SUBAPPLICATION NumericValue_TO_AR2_OPC (* VT-Eingabefeld (CInputNumber) UND OPC-UA (Remote) lesen, letzter Schreiber gewinnt (AR_LAST_2), als AR2 (bidirektional) an einen Consumer weiterreichen. Was der Consumer zurueckechot wird auf BEIDE Wege zurueckgemeldet (VT-Anzeige + Publish) *)
  (* Standard: 61499-2; Description: Copyright (c) 2026 Meisterschulen am Ostbahnhof This program and the accompanying materials are made available under the terms of the Eclipse Public License 2.0 which is available at https://www.eclipse.org/legal/epl-2.0/ SPDX-License-Identifier: EPL-2.0 *)
  (* Version 1.1, 2026-09-16, Franz Höpfinger, Meisterschulen am Ostbahnhof, Neuer optionaler Ausgangs-Plug VALUE_OUT ergaenzt (AR_SPLIT_2 zu AR_SPLIT_3, 3. Zweig = plain-AR-Spiegel von AR_TO_AR2.AR_OUT) - damit externe Consumer den aktuellen Wert lesen koennen, ohne selbst denselben OPC-UA-Knoten lokal zu abonnieren (FORTE: 'Cannot add another one'). Unverdrahtet lassen, wenn nicht gebraucht. Siehe BERICHT_2026-09-16_STG3_I1_I3_I4_I6_STALE_REMOTE_SUBSCRIBE.md Abschnitt 16-17 Gruppe C. *)
  (* Version 1.0, 2026-08-31, Franz Höpfinger, Meisterschulen am Ostbahnhof, VT+OPC-UA sibling of NumericValue_TO_AR2 (VT only) / OPC_TO_AR2 (OPC only) - merges both live sources via AR_LAST_2 (last writer wins), exactly like the VT/Web merge already proven in RampLimitFS_TO_logiBUS_QDA_PWM_OPC.SUB *)
  PACKAGE MyLib::sys;
  IMPORT isobus::UT::Q::const::IDs::ID_NULL;
  IMPORT logiBUS::utils::conversion::phys::NumericObjectPool_S;
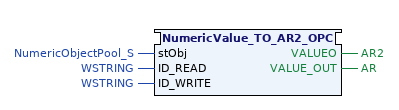
  VAR_INPUT
    stObj : logiBUS::utils::conversion::phys::NumericObjectPool_S := (u16ObjId := ID_NULL, r32Scale := 1.0, i32Offset := 0, u8Decimals := 0);
    ID_READ : WSTRING; (* Remote-Subscribe-Adresse (REAL, ACTION=SUBSCRIBE) *)
    ID_WRITE : WSTRING; (* Remote-Echo-Adresse (REAL, ACTION=PUBLISH) - meldet zurueck, was der Consumer gerade als aktuellen/persistierten Wert liefert *)
  END_VAR
  PLUGS
    VALUEO : adapter::types::bidirectional::AR2;
    VALUE_OUT : adapter::types::unidirectional::AR; (* Optional: plain-AR-Spiegel des aktuellen Werts (= AR_TO_AR2.AR_OUT), fuer externe Consumer statt eigenem lokalen OPC-UA-Self-Subscribe. Unverdrahtet lassen, wenn nicht gebraucht. *)
  END_PLUGS
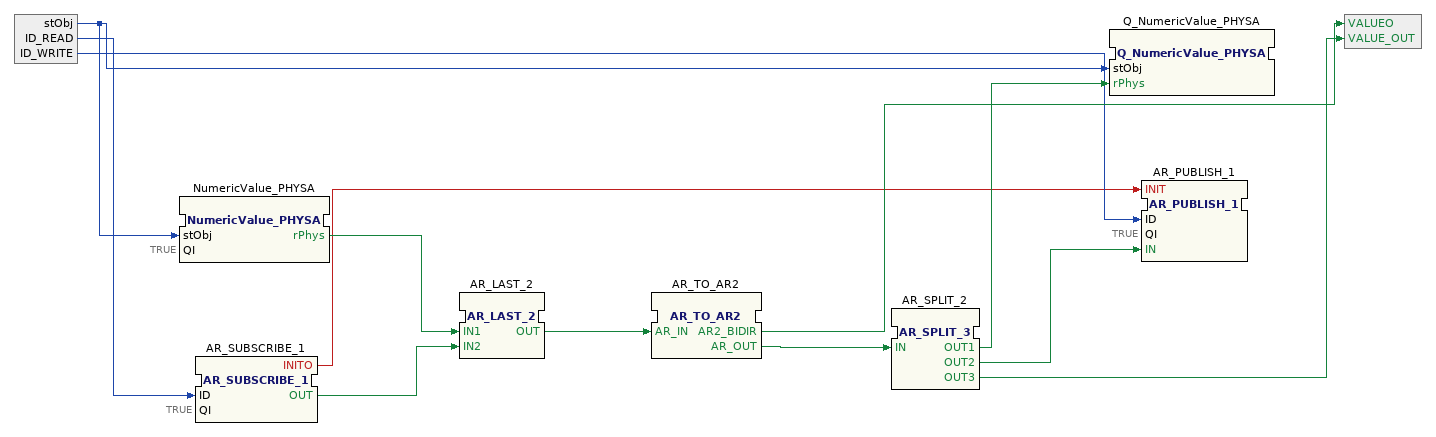
  FBS
    NumericValue_PHYSA : isobus::UT::io::NumericValue::NumericValue_PHYSA(QI := TRUE);
    AR_SUBSCRIBE_1 : adapter::net::AR_SUBSCRIBE_1(QI := TRUE);
    Q_NumericValue_PHYSA : isobus::UT::Q::Q_NumericValue_PHYSA;
    AR_PUBLISH_1 : adapter::net::AR_PUBLISH_1(QI := TRUE);
    AR_TO_AR2 : adapter::conversion::bidirectional::AR_TO_AR2;
    AR_SPLIT_2 : adapter::events::unidirectional::AR_SPLIT_3;
    AR_LAST_2 : adapter::events::unidirectional::AR_LAST_2;
  END_FBS
  EVENT_CONNECTIONS
    AR_SUBSCRIBE_1.INITO TO AR_PUBLISH_1.INIT;
  END_CONNECTIONS
  DATA_CONNECTIONS
    stObj TO NumericValue_PHYSA.stObj;
    stObj TO Q_NumericValue_PHYSA.stObj;
    ID_READ TO AR_SUBSCRIBE_1.ID;
    ID_WRITE TO AR_PUBLISH_1.ID;
  END_CONNECTIONS
  ADAPTER_CONNECTIONS
    AR_TO_AR2.AR2_BIDIR TO VALUEO;
    AR_TO_AR2.AR_OUT TO AR_SPLIT_2.IN;
    AR_SPLIT_2.OUT1 TO Q_NumericValue_PHYSA.rPhys;
    AR_SPLIT_2.OUT2 TO AR_PUBLISH_1.IN;
    AR_SPLIT_2.OUT3 TO VALUE_OUT;
    AR_LAST_2.OUT TO AR_TO_AR2.AR_IN;
    NumericValue_PHYSA.rPhys TO AR_LAST_2.IN1;
    AR_SUBSCRIBE_1.OUT TO AR_LAST_2.IN2;
  END_CONNECTIONS
END_SUBAPPLICATION
